// TwinCAT 3 PLC project Tc3EventLoggerUsage
// ProgramVersion: 3.1.4022.0
// libraries:
//   Tc2_Standard, * (Beckhoff Automation GmbH)
//   Tc2_System, * (Beckhoff Automation GmbH)
//   Tc2_Utilities, * (Beckhoff Automation GmbH)
//   Tc3_EventLogger, * (Beckhoff Automation GmbH)
//   Tc3_Module, * (Beckhoff Automation GmbH)
// project tree:
//   GVLs/ GVL.TcGVL
//   / PlcTask.TcTTO (not stored)
//   POUs/ FB_Control.TcPOU, FB_MathCalculation.TcPOU, MAIN.TcPOU
// real-time tasks:
//   TASK PlcTask: cycle T#10ms, priority 20, ADS port 350

// ---- GVLs/GVL.TcGVL
{attribute 'qualified_only'}
VAR_GLOBAL
	eEventTraceLevel : TcEventSeverity := TcEventSeverity.Critical;  
END_VAR

// ---- POUs/FB_Control.TcPOU
// encapsulation of FB_MathCalculation
FUNCTION_BLOCK FB_Control
VAR_INPUT
END_VAR
VAR_OUTPUT
	bError : BOOL;
	ipResultMessage : I_TcMessage := fbResult;
END_VAR

VAR
	fbResult : FB_TcMessage;
	fbSource : FB_TcSourceInfo;
	
	fDividend : LREAL := 42.0; 
	fDivisor : LREAL := 1.0; 
	fQuotient : LREAL;
	
	fbMath : FB_MathCalculation := (eTraceLevel:=TcEventSeverity.Critical); // nearly nothing of this internal FB should be logged 
	
	hrLastInternalError : HRESULT;
	
	 {attribute 'hide'}
	bOwnTL : BOOL; // own trace level is set
	 {attribute 'hide'} 
	eOwnTL : TcEventSeverity := TcEventSeverity.Critical;
END_VAR

// whether the event trace level is taken from the library default or not. This could be set via Online View too.
{attribute 'monitoring':='call'}
PROPERTY bTraceLevelDefault : BOOL
GET
bTraceLevelDefault := NOT bOwnTL;
END_GET
SET
bOwnTL := NOT bTraceLevelDefault;
END_SET
END_PROPERTY

// current trace level for this FB. This could be set via Online View too.
{attribute 'monitoring':='call'}
PROPERTY eTraceLevel : TcEventSeverity
GET
IF bOwnTL THEN
	eTraceLevel := eOwnTL;
ELSE
	eTraceLevel := GVL.eEventTraceLevel;
END_IF
END_GET
SET
bOwnTL := TRUE;
eOwnTL := eTraceLevel;
END_SET
END_PROPERTY

METHOD Execute
VAR_INPUT
END_VAR

VAR
	hr : HRESULT;
END_VAR
fbMath.Division(fDividend:=fDividend, fDivisor:=fDivisor, fQuotient:=fQuotient);

bError := fbMath.bError;
IF NOT fbResult.EqualsToEventEntryEx(stOther:=fbMath.ipResultMessage.stEventEntry) THEN
	fbSource.ResetToDefault();
	fbSource.ExtendName(sExtension:='.Execute() -> ');
	fbSource.ExtendName(sExtension:=fbMath.ipResultMessage.ipSourceInfo.sName);
	fbSource.ExtendName(sExtension:='.Division()');
	hr := fbResult.CreateEx(stEventEntry:=fbMath.ipResultMessage.stEventEntry, ipSourceInfo:=fbSource);
	IF FAILED(hr) THEN
		hrLastInternalError := hr;
	END_IF

	IF bError AND fbResult.eSeverity >= eTraceLevel THEN
		hr := fbResult.Send(0);
		IF FAILED(hr) THEN
			hrLastInternalError := hr;
		END_IF
	END_IF 
END_IF
END_METHOD

END_FUNCTION_BLOCK

// ---- POUs/FB_MathCalculation.TcPOU
FUNCTION_BLOCK FB_MathCalculation
VAR_INPUT
END_VAR
VAR_OUTPUT 
	bError : BOOL;
	ipResultMessage : I_TcMessage := fbResult;
END_VAR

VAR
	fbResult : FB_TcMessage;
(*	fbSource : FB_TcSourceInfo;	// optional *)
	
	hrLastInternalError : HRESULT;
	
	 {attribute 'hide'}
	bOwnTL : BOOL; // own trace level is set
	 {attribute 'hide'}
	eOwnTL : TcEventSeverity := TcEventSeverity.Critical;
END_VAR

// returns TRUE if succeeded
METHOD Addition : BOOL
VAR_INPUT
	nIn1 : UDINT;
	nIn2 : UDINT;
	nSum : REFERENCE TO UDINT;
END_VAR

VAR
	hr : HRESULT;
END_VAR
nSum := nIn1 + nIn2;

IF (nSum < nIn1) THEN // an overflow occurred
	bError := TRUE;

	IF NOT fbResult.EqualsToEventEntryEx(stOther:=TC_EVENTS.Win32EventClass.ERROR_ARITHMETIC_OVERFLOW) THEN
		hr := fbResult.CreateEx(TC_EVENTS.Win32EventClass.ERROR_ARITHMETIC_OVERFLOW, 0 ); //This uses dyn ressources and shouldn't be called cyclically.
		IF FAILED(hr) THEN
			hrLastInternalError := hr;
		END_IF
		
		IF fbResult.eSeverity >= eTraceLevel THEN
			hr := fbResult.Send(0);
			IF FAILED(hr) THEN
				hrLastInternalError := hr;
			END_IF
		END_IF 
	END_IF
	
ELSE
	Addition := TRUE;
	bError := FALSE;
	IF NOT fbResult.EqualsToEventEntryEx(stOther:=SUCCESS_EVENT) THEN
		hr := fbResult.CreateEx(SUCCESS_EVENT, 0 ); //This uses dyn ressources and shouldn't be called cyclically.
		IF FAILED(hr) THEN
			hrLastInternalError := hr;
		END_IF
	END_IF
	
END_IF
END_METHOD

// whether the event trace level is taken from the library default or not. This could be set via Online View too.
{attribute 'monitoring':='call'}
PROPERTY bTraceLevelDefault : BOOL
GET
bTraceLevelDefault := NOT bOwnTL;
END_GET
SET
bOwnTL := NOT bTraceLevelDefault;
END_SET
END_PROPERTY

// returns TRUE if succeeded
METHOD Division : BOOL
VAR_INPUT
	fDividend : LREAL;
	fDivisor  : LREAL;
	fQuotient : REFERENCE TO LREAL;
END_VAR

VAR
	hr : HRESULT;
END_VAR
IF (fDivisor = 0) THEN
	bError := TRUE;
	//adapt source name if required (default is ads symbol name)
	//fbSource.Clear();
	//fbSource.sName := 'Math Calculation';
	IF NOT fbResult.EqualsToEventEntryEx(stOther:=TC_EVENTS.CalculationEventClass.DivisionByZero) THEN
		hr := fbResult.CreateEx(TC_EVENTS.CalculationEventClass.DivisionByZero, 0 (*fbSource*) ); //This uses dyn ressources and shouldn't be called cyclically.
		IF FAILED(hr) THEN
			hrLastInternalError := hr;
		END_IF
		//set Arguments if required
		//fbResult.ipArguments.Clear().Add ...
		//set JSON attribute if required
		//fbResult.SetJsonAttribute('{"DivionByZero":1,"Divisor":0}');
		
		IF fbResult.eSeverity >= eTraceLevel THEN
			hr := fbResult.Send(0);
			IF FAILED(hr) THEN
				hrLastInternalError := hr;
			END_IF
		END_IF 
	END_IF
	
ELSE
	fQuotient := fDividend / fDivisor;
	Division := TRUE;
	bError := FALSE;
	IF NOT fbResult.EqualsToEventEntryEx(stOther:=SUCCESS_EVENT) THEN
		hr := fbResult.CreateEx(SUCCESS_EVENT, 0 (*fbSource*) ); //This uses dyn ressources and shouldn't be called cyclically.
		IF FAILED(hr) THEN
			hrLastInternalError := hr;
		END_IF
	END_IF
	
END_IF
END_METHOD

// current trace level for this FB. This could be set via Online View too. 
{attribute 'monitoring':='call'}
PROPERTY eTraceLevel : TcEventSeverity
GET
IF bOwnTL THEN
	eTraceLevel := eOwnTL;
ELSE
	eTraceLevel := GVL.eEventTraceLevel;
END_IF
END_GET
SET
bOwnTL := TRUE;
eOwnTL := eTraceLevel;
END_SET
END_PROPERTY

END_FUNCTION_BLOCK

// ---- POUs/MAIN.TcPOU
PROGRAM MAIN
VAR
	nState : USINT := 0;

	fDividend : LREAL := 42.0; 
	fDivisor : LREAL := 1.0; // set to zero to force an error
	fQuotient : LREAL;
	
	// application POU using the result message interface to specify occurred errors (e.g. division by zero)
	fbMath : FB_MathCalculation := (eTraceLevel:=TcEventSeverity.Verbose); 
	
	// another application POU which encapsulates FB_MathCalculation
	fbCtrl : FB_Control := (eTraceLevel:=TcEventSeverity.Verbose); 
	
	sErrorText : STRING(255);
	bGetText : BOOL;
END_VAR

CASE nState OF
0: // calculation with fbMath
	fbMath.Division(fDividend:=fDividend, fDivisor:=fDivisor, fQuotient:=fQuotient);
	IF fbMath.bError THEN
		// error handling
		nState := 10;
	END_IF
	
1: // calculation with fbCtrl
	fbCtrl.Execute();
	IF fbCtrl.bError THEN
		// error handling
		// e.g. error text could be requested if execution failed.
		bGetText := TRUE;
		nState := 10;
	END_IF
	
10: // error occurred
	IF bGetText THEN
		IF fbCtrl.ipResultMessage.RequestEventText(	nLangId:=Tc3_EventLogger.GVL.nLangId_OnlineMonitoring, 
													sResult:=sErrorText, nResultSize:=SIZEOF(sErrorText) ) THEN
			bGetText := FALSE;
		END_IF
	END_IF
	
END_CASE

END_PROGRAM
